(* PLC project OOP_Curso, Beckhoff Automation GmbH TwinCAT PLC Control 3.5.13.21 *)
(* stored: creationDateTime 2023-03-05T21:09:17.8155442, modificationDateTime 2023-03-05T21:09:17.8155442 *)

TYPE ST_Property :
STRUCT
	b1,b2,b3 : BOOL;
	r1,r2,r3 : REAL;
	
END_STRUCT
END_TYPE

PROGRAM _06_Propiedad
VAR
	myFBProperty : FB_Ejemplo_Propiedad;
	
	bSet1, bSet2 : BOOL;
	
	IntData : INT;
	BoolData : BOOL;
	GetSTData : ST_Property;
	SetSTData : ST_Property;
	ioData    : INT;
	counter   : INT;
END_VAR

            IF bSet1 THEN
	bSet1:= FALSE;
	myFBProperty.ValueBool := TRUE;
	myFBProperty.ValueInt := 123;
	SetSTData.b1 := TRUE;
	SetSTData.b2 := FALSE;
	SetSTData.b3 := FALSE;
	SetSTData.r1 := 1.0;
	SetSTData.r2 := 2.0;
	SetSTData.r3 := 3.0;

END_IF

IF bSet2 THEN
	bSet2:= FALSE;
	myFBProperty.ValueBool := FALSE;
	myFBProperty.ValueInt := 456;
	SetSTData.b1 := FALSE;
	SetSTData.b2 := TRUE;
	SetSTData.b3 := TRUE;
	SetSTData.r1 := 11.0;
	SetSTData.r2 := 22.0;
	SetSTData.r3 := 33.0;
END_IF


IntData := 	myFBProperty.ValueInt;
BoolData := myFBProperty.ValueBool;

//STRUCT
GetSTData.b1 := myFBProperty.ValueST.b1;
GetSTData.r1 := myFBProperty.ValueST.r1;

myFBProperty.ValueST := SetSTData;

//IN_OUT;
IF counter < 0 OR counter > 9999 THEN
	counter := 1;
ELSE
	counter := counter + 1;
END_IF

//myFBProperty(myIN_OUT:=counter);
//myFBProperty.Value_INT_OUT := 120;
ioData := myFBProperty.Value_INT_OUT;
myFBProperty(myIN_OUT:=counter);
          
END_PROGRAM

FUNCTION_BLOCK FB_ejemplo_Propiedad
VAR_INPUT
END_VAR
VAR_OUTPUT
END_VAR
VAR_IN_OUT
	myIN_OUT : INT;
END_VAR
VAR
	myBool : BOOL;
	myInt : INT;
	myST  : ST_Property;
END_VAR

            
          

PROPERTY ValueBool : BOOL
GET
VAR
END_VAR
                    ValueBool := myBool;
                  
END_GET
SET
VAR
END_VAR
                     myBool := ValueBool;
                  
END_SET
END_PROPERTY

PROPERTY ValueInt : INT
GET
VAR
END_VAR
                    ValueInt := myint;
                  
END_GET
SET
VAR
END_VAR
                     myint := ValueInt;
                  
END_SET
END_PROPERTY

PROPERTY ValueST : reference to ST_Property
GET
VAR
END_VAR
                    ValueST REF= myST;
                  
END_GET
SET
VAR
END_VAR
                    IF NOT __ISVALIDREF(myIN_OUT) THEN
	RETURN;
END_IF

myST := ValueST;
                  
END_SET
END_PROPERTY

PROPERTY Value_INT_OUT : INT
GET
VAR
END_VAR
                    IF NOT __ISVALIDREF(myIN_OUT) THEN
	RETURN;
END_IF

Value_INT_OUT := myIN_OUT;
                  
END_GET
SET
VAR
END_VAR
                    myIN_OUT := Value_INT_OUT;
                  
END_SET
END_PROPERTY
END_FUNCTION_BLOCK
